(*
SPDX-FileCopyrightText: © 2026 Oleksandr Tiutyk <trofimich@gmail.com>
SPDX-License-Identifier: MIT
License: https://opensource.org/license/mit
*)

INTERFACE IGeneralException EXTENDS IException

{attribute 'monitoring' := 'call'}
PROPERTY FINAL ErrorCode : UDINT
GET
END_GET
END_PROPERTY

METHOD GetRootException : IException
END_METHOD

{attribute 'monitoring' := 'call'}
PROPERTY FINAL InnerException : IException
GET
END_GET
END_PROPERTY

{attribute 'monitoring' := 'call'}
PROPERTY FINAL SourceMessage : REFERENCE TO ERROR_MESSAGE
GET
END_GET
END_PROPERTY

END_INTERFACE

(* stored: Version 1.1.0.1
   Itf IGeneralException: Id {d983ee74-5791-40d6-b742-92434317edb5}
   Property ErrorCode: Id {6b64a45c-051a-48ee-a27d-c3dbcc60e4bf}
   Get Get: Id {04d5d64f-d327-43d7-9f8a-41fb2f21cb91}
   Method GetRootException: Id {d1541aef-c327-42c5-8db6-0308e8de7f5b}
   Property InnerException: Id {b22600ff-32e1-412a-9999-be966eb3f9a6}
   Get Get: Id {31d5db1b-8b93-413d-8924-a82a16beeb43}
   Property SourceMessage: Id {5e4316d5-0fc4-47ec-9091-572b6a8bd406}
   Get Get: Id {84e53f69-0a0a-48fb-8362-a2dbf733bd49} *)
